   // One irrigation event is a volume-bounded batch. The pre-flush and
   // post-flush sections use only carrier water; metering pumps run only in
   // the middle FERTIGATE section. A zero volume SP preserves continuous
   // manual commissioning behavior.
   #Pre_Flush_Ratio_Limited := "DB1".Pre_Flush_Ratio;
   IF #Pre_Flush_Ratio_Limited < 0.0 THEN #Pre_Flush_Ratio_Limited := 0.0; END_IF;
   IF #Pre_Flush_Ratio_Limited > 1.0 THEN #Pre_Flush_Ratio_Limited := 1.0; END_IF;
   #Post_Flush_Ratio_Limited := "DB1".Post_Flush_Ratio;
   IF #Post_Flush_Ratio_Limited < 0.0 THEN #Post_Flush_Ratio_Limited := 0.0; END_IF;
   IF #Post_Flush_Ratio_Limited > (1.0 - #Pre_Flush_Ratio_Limited) THEN
      #Post_Flush_Ratio_Limited := 1.0 - #Pre_Flush_Ratio_Limited;
   END_IF;
   "DB1".Pre_Flush_Volume := "DB1".Water_Volume_SP * #Pre_Flush_Ratio_Limited;
   "DB1".Fertigation_End_Volume := "DB1".Water_Volume_SP
      * (1.0 - #Post_Flush_Ratio_Limited);
   "DB1".Batch_Fertigation_Active := FALSE;
   "DB1".Water_Batch_Active := FALSE;

   IF "DB1".Water_Enable < 0.5 THEN
      IF "DB1".Water_Volume_Complete THEN
         "DB1".Water_Batch_Phase := 4;
      ELSE
         "DB1".Water_Batch_Phase := 0;
      END_IF;
   ELSIF "DB1".Water_Volume_Complete THEN
      "DB1".Water_Batch_Phase := 4;
   ELSIF "DB1".Water_Volume_SP <= 0.0 THEN
      "DB1".Water_Batch_Phase := 2;
      "DB1".Water_Batch_Active := TRUE;
      "DB1".Batch_Fertigation_Active := "DB1".Water_Flow_OK;
   ELSIF "DB1".Water_Volume_Actual < "DB1".Pre_Flush_Volume THEN
      "DB1".Water_Batch_Phase := 1;
      "DB1".Water_Batch_Active := TRUE;
   ELSIF "DB1".Water_Volume_Actual < "DB1".Fertigation_End_Volume THEN
      "DB1".Water_Batch_Phase := 2;
      "DB1".Water_Batch_Active := TRUE;
      "DB1".Batch_Fertigation_Active := "DB1".Water_Flow_OK;
   ELSE
      "DB1".Water_Batch_Phase := 3;
      "DB1".Water_Batch_Active := TRUE;
   END_IF;

   // Scheme B: independent N, P, K and acid metering pumps.
   // Execution_Enable is FALSE by default, so legacy simulation behavior is isolated.
   "DB_Pump_N"(
      Enable := "DB_Actuator".Execution_Enable AND "DB1".Batch_Fertigation_Active
         AND NOT "DB1".Emergency_Stop,
      Flow_SP := "DB1".q_n_cmd,
      Flow_PV := "DB_Actuator".N_Flow_PV,
      Flow_Min := "DB_Actuator".N_Flow_Min,
      Flow_Max := "DB_Actuator".N_Flow_Max,
      AO_Off_Raw := "DB_Actuator".N_AO_Off_Raw,
      AO_Raw_Min := "DB_Actuator".N_AO_Raw_Min,
      AO_Raw_Max := "DB_Actuator".N_AO_Raw_Max,
      Kp_Flow := "DB_Actuator".N_Kp_Flow,
      Ki_Flow := "DB_Actuator".N_Ki_Flow,
      Cycle_Time_s := "DB_Actuator".Cycle_Time_s,
      Run_Feedback := "DB_Actuator".N_Run_Feedback,
      Drive_Ready := "DB_Actuator".N_Drive_Ready,
      Drive_Fault := "DB_Actuator".N_Drive_Fault,
      Tank_Low_Level := "DB_Actuator".N_Tank_Low_Level,
      Water_Flow_OK := "DB_Actuator".Water_Flow_OK,
      Reset := "DB_Actuator".Reset_All OR "DB_Actuator".N_Reset,
      Start_Fail_Delay_s := "DB_Actuator".N_Start_Fail_Delay_s,
      No_Flow_Delay_s := "DB_Actuator".N_No_Flow_Delay_s,
      Flow_Deviation_Delay_s := "DB_Actuator".N_Flow_Deviation_Delay_s,
      No_Flow_Threshold := "DB_Actuator".N_No_Flow_Threshold,
      Flow_Deviation_Abs := "DB_Actuator".N_Flow_Deviation_Abs,
      Flow_Deviation_Rel := "DB_Actuator".N_Flow_Deviation_Rel,
      Run_Command => "DB_Actuator".N_Run_Command,
      AO_Command_Raw => "DB_Actuator".N_AO_Command_Raw,
      Flow_SP_Limited => "DB_Actuator".N_Flow_SP_Limited,
      Running => "DB_Actuator".N_Running,
      Ready => "DB_Actuator".N_Ready,
      No_Flow_Alarm => "DB_Actuator".N_No_Flow_Alarm,
      Flow_Deviation_Alarm => "DB_Actuator".N_Flow_Deviation_Alarm,
      Start_Fail_Alarm => "DB_Actuator".N_Start_Fail_Alarm,
      Saturated => "DB_Actuator".N_Saturated,
      Interlocked => "DB_Actuator".N_Interlocked,
      Control_Percent => "DB_Actuator".N_Control_Percent
   );

   "DB_Pump_P"(
      Enable := "DB_Actuator".Execution_Enable AND "DB1".Batch_Fertigation_Active
         AND NOT "DB1".Emergency_Stop,
      Flow_SP := "DB1".q_p_cmd,
      Flow_PV := "DB_Actuator".P_Flow_PV,
      Flow_Min := "DB_Actuator".P_Flow_Min,
      Flow_Max := "DB_Actuator".P_Flow_Max,
      AO_Off_Raw := "DB_Actuator".P_AO_Off_Raw,
      AO_Raw_Min := "DB_Actuator".P_AO_Raw_Min,
      AO_Raw_Max := "DB_Actuator".P_AO_Raw_Max,
      Kp_Flow := "DB_Actuator".P_Kp_Flow,
      Ki_Flow := "DB_Actuator".P_Ki_Flow,
      Cycle_Time_s := "DB_Actuator".Cycle_Time_s,
      Run_Feedback := "DB_Actuator".P_Run_Feedback,
      Drive_Ready := "DB_Actuator".P_Drive_Ready,
      Drive_Fault := "DB_Actuator".P_Drive_Fault,
      Tank_Low_Level := "DB_Actuator".P_Tank_Low_Level,
      Water_Flow_OK := "DB_Actuator".Water_Flow_OK,
      Reset := "DB_Actuator".Reset_All OR "DB_Actuator".P_Reset,
      Start_Fail_Delay_s := "DB_Actuator".P_Start_Fail_Delay_s,
      No_Flow_Delay_s := "DB_Actuator".P_No_Flow_Delay_s,
      Flow_Deviation_Delay_s := "DB_Actuator".P_Flow_Deviation_Delay_s,
      No_Flow_Threshold := "DB_Actuator".P_No_Flow_Threshold,
      Flow_Deviation_Abs := "DB_Actuator".P_Flow_Deviation_Abs,
      Flow_Deviation_Rel := "DB_Actuator".P_Flow_Deviation_Rel,
      Run_Command => "DB_Actuator".P_Run_Command,
      AO_Command_Raw => "DB_Actuator".P_AO_Command_Raw,
      Flow_SP_Limited => "DB_Actuator".P_Flow_SP_Limited,
      Running => "DB_Actuator".P_Running,
      Ready => "DB_Actuator".P_Ready,
      No_Flow_Alarm => "DB_Actuator".P_No_Flow_Alarm,
      Flow_Deviation_Alarm => "DB_Actuator".P_Flow_Deviation_Alarm,
      Start_Fail_Alarm => "DB_Actuator".P_Start_Fail_Alarm,
      Saturated => "DB_Actuator".P_Saturated,
      Interlocked => "DB_Actuator".P_Interlocked,
      Control_Percent => "DB_Actuator".P_Control_Percent
   );

   "DB_Pump_K"(
      Enable := "DB_Actuator".Execution_Enable AND "DB1".Batch_Fertigation_Active
         AND NOT "DB1".Emergency_Stop,
      Flow_SP := "DB1".q_k_cmd,
      Flow_PV := "DB_Actuator".K_Flow_PV,
      Flow_Min := "DB_Actuator".K_Flow_Min,
      Flow_Max := "DB_Actuator".K_Flow_Max,
      AO_Off_Raw := "DB_Actuator".K_AO_Off_Raw,
      AO_Raw_Min := "DB_Actuator".K_AO_Raw_Min,
      AO_Raw_Max := "DB_Actuator".K_AO_Raw_Max,
      Kp_Flow := "DB_Actuator".K_Kp_Flow,
      Ki_Flow := "DB_Actuator".K_Ki_Flow,
      Cycle_Time_s := "DB_Actuator".Cycle_Time_s,
      Run_Feedback := "DB_Actuator".K_Run_Feedback,
      Drive_Ready := "DB_Actuator".K_Drive_Ready,
      Drive_Fault := "DB_Actuator".K_Drive_Fault,
      Tank_Low_Level := "DB_Actuator".K_Tank_Low_Level,
      Water_Flow_OK := "DB_Actuator".Water_Flow_OK,
      Reset := "DB_Actuator".Reset_All OR "DB_Actuator".K_Reset,
      Start_Fail_Delay_s := "DB_Actuator".K_Start_Fail_Delay_s,
      No_Flow_Delay_s := "DB_Actuator".K_No_Flow_Delay_s,
      Flow_Deviation_Delay_s := "DB_Actuator".K_Flow_Deviation_Delay_s,
      No_Flow_Threshold := "DB_Actuator".K_No_Flow_Threshold,
      Flow_Deviation_Abs := "DB_Actuator".K_Flow_Deviation_Abs,
      Flow_Deviation_Rel := "DB_Actuator".K_Flow_Deviation_Rel,
      Run_Command => "DB_Actuator".K_Run_Command,
      AO_Command_Raw => "DB_Actuator".K_AO_Command_Raw,
      Flow_SP_Limited => "DB_Actuator".K_Flow_SP_Limited,
      Running => "DB_Actuator".K_Running,
      Ready => "DB_Actuator".K_Ready,
      No_Flow_Alarm => "DB_Actuator".K_No_Flow_Alarm,
      Flow_Deviation_Alarm => "DB_Actuator".K_Flow_Deviation_Alarm,
      Start_Fail_Alarm => "DB_Actuator".K_Start_Fail_Alarm,
      Saturated => "DB_Actuator".K_Saturated,
      Interlocked => "DB_Actuator".K_Interlocked,
      Control_Percent => "DB_Actuator".K_Control_Percent
   );

   "DB_Pump_Acid"(
      Enable := "DB_Actuator".Execution_Enable AND "DB1".Batch_Fertigation_Active
         AND NOT "DB1".Emergency_Stop,
      Flow_SP := "DB1".q_a_cmd,
      Flow_PV := "DB_Actuator".Acid_Flow_PV,
      Flow_Min := "DB_Actuator".Acid_Flow_Min,
      Flow_Max := "DB_Actuator".Acid_Flow_Max,
      AO_Off_Raw := "DB_Actuator".Acid_AO_Off_Raw,
      AO_Raw_Min := "DB_Actuator".Acid_AO_Raw_Min,
      AO_Raw_Max := "DB_Actuator".Acid_AO_Raw_Max,
      Kp_Flow := "DB_Actuator".Acid_Kp_Flow,
      Ki_Flow := "DB_Actuator".Acid_Ki_Flow,
      Cycle_Time_s := "DB_Actuator".Cycle_Time_s,
      Run_Feedback := "DB_Actuator".Acid_Run_Feedback,
      Drive_Ready := "DB_Actuator".Acid_Drive_Ready,
      Drive_Fault := "DB_Actuator".Acid_Drive_Fault,
      Tank_Low_Level := "DB_Actuator".Acid_Tank_Low_Level,
      Water_Flow_OK := "DB_Actuator".Water_Flow_OK,
      Reset := "DB_Actuator".Reset_All OR "DB_Actuator".Acid_Reset,
      Start_Fail_Delay_s := "DB_Actuator".Acid_Start_Fail_Delay_s,
      No_Flow_Delay_s := "DB_Actuator".Acid_No_Flow_Delay_s,
      Flow_Deviation_Delay_s := "DB_Actuator".Acid_Flow_Deviation_Delay_s,
      No_Flow_Threshold := "DB_Actuator".Acid_No_Flow_Threshold,
      Flow_Deviation_Abs := "DB_Actuator".Acid_Flow_Deviation_Abs,
      Flow_Deviation_Rel := "DB_Actuator".Acid_Flow_Deviation_Rel,
      Run_Command => "DB_Actuator".Acid_Run_Command,
      AO_Command_Raw => "DB_Actuator".Acid_AO_Command_Raw,
      Flow_SP_Limited => "DB_Actuator".Acid_Flow_SP_Limited,
      Running => "DB_Actuator".Acid_Running,
      Ready => "DB_Actuator".Acid_Ready,
      No_Flow_Alarm => "DB_Actuator".Acid_No_Flow_Alarm,
      Flow_Deviation_Alarm => "DB_Actuator".Acid_Flow_Deviation_Alarm,
      Start_Fail_Alarm => "DB_Actuator".Acid_Start_Fail_Alarm,
      Saturated => "DB_Actuator".Acid_Saturated,
      Interlocked => "DB_Actuator".Acid_Interlocked,
      Control_Percent => "DB_Actuator".Acid_Control_Percent
   );

   "DB_Actuator".Any_Demand := "DB_Actuator".Execution_Enable
      AND "DB1".Batch_Fertigation_Active AND (
      ("DB1".q_n_cmd > 0.0) OR ("DB1".q_p_cmd > 0.0)
      OR ("DB1".q_k_cmd > 0.0) OR ("DB1".q_a_cmd > 0.0));

   "DB_Actuator".Any_Trip := "DB_Actuator".Execution_Enable AND (
      "DB1".Water_Pump_Fault
      OR
      "DB_Actuator".N_Start_Fail_Alarm OR "DB_Actuator".N_No_Flow_Alarm
      OR "DB_Actuator".P_Start_Fail_Alarm OR "DB_Actuator".P_No_Flow_Alarm
      OR "DB_Actuator".K_Start_Fail_Alarm OR "DB_Actuator".K_No_Flow_Alarm
      OR "DB_Actuator".Acid_Start_Fail_Alarm OR "DB_Actuator".Acid_No_Flow_Alarm
      OR "DB_Actuator".N_Drive_Fault OR "DB_Actuator".P_Drive_Fault
      OR "DB_Actuator".K_Drive_Fault OR "DB_Actuator".Acid_Drive_Fault
      OR "DB_Actuator".N_Tank_Low_Level OR "DB_Actuator".P_Tank_Low_Level
      OR "DB_Actuator".K_Tank_Low_Level OR "DB_Actuator".Acid_Tank_Low_Level
      OR ("DB_Actuator".Any_Demand AND NOT "DB_Actuator".Water_Flow_OK));

   "DB_Actuator".Any_Alarm := "DB_Actuator".Execution_Enable AND (
      "DB_Actuator".Any_Trip OR "DB1".Water_Pump_Alarm
      OR "DB_Actuator".N_Flow_Deviation_Alarm
      OR "DB_Actuator".P_Flow_Deviation_Alarm
      OR "DB_Actuator".K_Flow_Deviation_Alarm
      OR "DB_Actuator".Acid_Flow_Deviation_Alarm);

   "DB1".Actuator_Execution_Enable := "DB_Actuator".Execution_Enable;
   "DB1".Actuator_Any_Alarm := "DB_Actuator".Any_Alarm;
   "DB1".Actuator_Any_Trip := "DB_Actuator".Any_Trip;

   IF "DB_Actuator".Execution_Enable THEN
      // The total fertilizer AO is forced off in Scheme B to prevent double dosing.
      "DB1".AQ_Valve_F_Raw := 0;
      "DB1".AQ_Valve_N_Raw := "DB_Actuator".N_AO_Command_Raw;
      "DB1".AQ_Valve_P_Raw := "DB_Actuator".P_AO_Command_Raw;
      "DB1".AQ_Valve_K_Raw := "DB_Actuator".K_AO_Command_Raw;
      "DB1".AQ_Valve_A_Raw := "DB_Actuator".Acid_AO_Command_Raw;

      // Real feedback replaces the previous command-as-feedback simulation value.
      "DB1".Valve_F_Actual := "DB_Actuator".N_Flow_PV
         + "DB_Actuator".P_Flow_PV + "DB_Actuator".K_Flow_PV;
      "DB1".Valve_A_Actual := "DB_Actuator".Acid_Flow_PV;
   END_IF;

   IF "DB1".System_Alarm_Reset THEN
      "DB1".System_Alarm_Light := FALSE;
   END_IF;
   IF "DB_Actuator".Any_Alarm THEN
      "DB1".System_Alarm_Light := TRUE;
   END_IF;
END_FUNCTION

FUNCTION "FC_CallFertigationControl" : Void
{ S7_Optimized_Access := 'TRUE' }
VERSION : 0.1
   VAR_TEMP
      Mode_EStop : Bool;
      Mode_Manual : Bool;
      Mode_Remote_Auto : Bool;
      Mode_Stage_Auto : Bool;
      Mode_Local_Auto : Bool;
      Mode_Standby : Bool;
      Remote_Auto_Available : Bool;
      PID_Control_Enable : Bool;
      Gain_Desired_Point : Int;
      Gain_q_f_Estimate : Real;
      Effective_Decoupler_Enable : Bool;
      Control_CycleTime : Real;
   END_VAR

BEGIN
   // 在 OB1 中调用本 FC，即可完成：
   // DB1 输入区 -> FB_FertigationControl -> DB1 输出区。
   // 固定模式表：
   // 1) Emergency_Stop=TRUE -> 急停，所有输出归零。
   // 2) Emergency_Stop=FALSE 且 Manual_Mode=TRUE -> 手动直接流量输出。
   // 3) Emergency_Stop=FALSE 且 Manual_Mode=FALSE 且 Auto_Mode=TRUE 且 SAC_Enable=TRUE -> 远程自动。
   // 4) Emergency_Stop=FALSE 且 Manual_Mode=FALSE 且 Auto_Mode=TRUE 且 SAC_Enable=FALSE 且 Stage_Auto_SP_Enable=TRUE -> 阶段自动。
   // 5) Emergency_Stop=FALSE 且 Manual_Mode=FALSE 且 Auto_Mode=TRUE 且 SAC_Enable=FALSE 且 Stage_Auto_SP_Enable=FALSE -> 本地定值自动。
   // 6) Emergency_Stop=FALSE 且 Manual_Mode=FALSE 且 Auto_Mode=FALSE -> 待机，所有输出归零。
   // 开关量联锁和报警灯由 FC_ModeInterlock_LAD 完成。
   // 六种互斥运行模式由 FC_ModeSelector_LAD 完成。
   // 连续量限幅、斜坡、模拟量换算和自动控制算法保留在 SCL。

   "FC_ModeInterlock_LAD"();

   // 远程命令只有在心跳正常时才有效；失联后把 SAC 请求视为无效，
   // 由现有 LAD 模式表自动选择阶段自动或本地定值自动。
   IF NOT "DB1".Remote_Comms_OK THEN
      "DB1".SAC_Enable := FALSE;
   END_IF;
   // 自动模式的本地来源固定为生长阶段目标，不提供人工来源切换。
   "DB1".Stage_Auto_SP_Enable := TRUE;
   #Remote_Auto_Available := "DB1".SAC_Enable AND "DB1".Remote_Comms_OK;

   "FC_ModeSelector_LAD"(
      Emergency_Stop := "DB1".Emergency_Stop,
      Manual_Mode := "DB1".Manual_Mode,
      Auto_Mode := "DB1".Auto_Mode,
      SAC_Enable := #Remote_Auto_Available,
      Stage_Auto_SP_Enable := "DB1".Stage_Auto_SP_Enable,
      Mode_EStop => #Mode_EStop,
      Mode_Manual => #Mode_Manual,
      Mode_Remote_Auto => #Mode_Remote_Auto,
      Mode_Stage_Auto => #Mode_Stage_Auto,
      Mode_Local_Auto => #Mode_Local_Auto,
      Mode_Standby => #Mode_Standby
   );

   // Manual_Active, Auto_Active, Manual_PumpValve_Enable and the two manual
   // flow selections are discrete interlocks owned by FC_ModeInterlock_LAD.
   // Do not assign them again in SCL; one tag must have one logic owner.

   #PID_Control_Enable := #Mode_Manual OR #Mode_Remote_Auto OR #Mode_Stage_Auto OR #Mode_Local_Auto;

   // PLC-native low/medium/high gain schedule. Python only commissions the
   // table; normal selection, hysteresis and bumpless handoff run in the CPU.
   "DB1".Gain_Schedule_Valid := "DB1".Gain_Low_Valid
      AND "DB1".Gain_Mid_Valid AND "DB1".Gain_High_Valid
      AND ("DB1".Gain_Low_G_EC_F > 0.000001) AND ("DB1".Gain_Low_G_pH_A < -0.000001)
      AND ("DB1".Gain_Mid_G_EC_F > 0.000001) AND ("DB1".Gain_Mid_G_pH_A < -0.000001)
      AND ("DB1".Gain_High_G_EC_F > 0.000001) AND ("DB1".Gain_High_G_pH_A < -0.000001)
      AND ("DB1".Gain_Low_EC_SP > 0.0)
      AND ("DB1".Gain_Mid_EC_SP > 0.0)
      AND ("DB1".Gain_High_EC_SP > 0.0)
      AND ("DB1".Gain_Low_q_f < "DB1".Gain_Mid_q_f)
      AND ("DB1".Gain_Mid_q_f < "DB1".Gain_High_q_f)
      AND ("DB1".Gain_LM_Threshold < "DB1".Gain_MH_Threshold)
      AND ("DB1".Gain_Schedule_Hysteresis >= 0.0)
      AND ("DB1".Gain_Min_Hold_s >= 0.0);

   IF ("DB1".EC_Set_SP > 0.0) AND ("DB1".EC_Set_SP < 34.0) THEN
      #Gain_q_f_Estimate := ("DB1".EC_Set_SP * 136.0) / (35.0 - "DB1".EC_Set_SP);
   ELSE
      #Gain_q_f_Estimate := 0.0;
   END_IF;
   IF ("DB1".Gain_Point_Override >= 0) AND ("DB1".Gain_Point_Override <= 2) THEN
      #Gain_Desired_Point := "DB1".Gain_Point_Override;
   ELSIF "DB1".Active_Gain_Point = 0 THEN
      IF #Gain_q_f_Estimate > ("DB1".Gain_LM_Threshold + "DB1".Gain_Schedule_Hysteresis) THEN
         #Gain_Desired_Point := 1;
      ELSE
         #Gain_Desired_Point := 0;
      END_IF;
   ELSIF "DB1".Active_Gain_Point = 2 THEN
      IF #Gain_q_f_Estimate < ("DB1".Gain_MH_Threshold - "DB1".Gain_Schedule_Hysteresis) THEN
         #Gain_Desired_Point := 1;
      ELSE
         #Gain_Desired_Point := 2;
      END_IF;
   ELSE
      IF #Gain_q_f_Estimate < ("DB1".Gain_LM_Threshold - "DB1".Gain_Schedule_Hysteresis) THEN
         #Gain_Desired_Point := 0;
      ELSIF #Gain_q_f_Estimate > ("DB1".Gain_MH_Threshold + "DB1".Gain_Schedule_Hysteresis) THEN
         #Gain_Desired_Point := 2;
      ELSE
         #Gain_Desired_Point := 1;
      END_IF;
   END_IF;

   IF "DB1".Gain_Schedule_Enable AND "DB1".Gain_Schedule_Valid THEN
      IF "DB1".Gain_Hold_Elapsed_s < 3600.0 THEN
         "DB1".Gain_Hold_Elapsed_s := "DB1".Gain_Hold_Elapsed_s + 0.1;
      END_IF;
      IF "DB1".Active_Gain_Point < 0 THEN
         "DB1".Gain_Switch_Pending := TRUE;
      ELSIF (#Gain_Desired_Point <> "DB1".Active_Gain_Point)
         AND ("DB1".Gain_Hold_Elapsed_s >= "DB1".Gain_Min_Hold_s) THEN
         "DB1".Gain_Switch_Pending := TRUE;
      END_IF;

      // Pending makes the effective enable FALSE below. The FB ramps its
      // applied weight to zero before this block replaces the active matrix.
      IF "DB1".Gain_Switch_Pending AND ("DB1".Decoupler_Weight_Applied <= 0.01) THEN
         IF #Gain_Desired_Point = 0 THEN
            "DB1".G_EC_F := "DB1".Gain_Low_G_EC_F;
            "DB1".G_EC_A := "DB1".Gain_Low_G_EC_A;
            "DB1".G_pH_F := "DB1".Gain_Low_G_pH_F;
            "DB1".G_pH_A := "DB1".Gain_Low_G_pH_A;
            "DB1".IMC_Tau_EC_s := "DB1".Gain_Low_Tau_s;
            "DB1".IMC_Delay_s := "DB1".Gain_Low_Delay_s;
            "DB1".Mixing_Delay_s := "DB1".Gain_Low_Delay_s;
            "DB1".Active_Gain_EC_SP := "DB1".Gain_Low_EC_SP;
            "DB1".Active_Gain_q_f := "DB1".Gain_Low_q_f;
         ELSIF #Gain_Desired_Point = 1 THEN
            "DB1".G_EC_F := "DB1".Gain_Mid_G_EC_F;
            "DB1".G_EC_A := "DB1".Gain_Mid_G_EC_A;
            "DB1".G_pH_F := "DB1".Gain_Mid_G_pH_F;
            "DB1".G_pH_A := "DB1".Gain_Mid_G_pH_A;
            "DB1".IMC_Tau_EC_s := "DB1".Gain_Mid_Tau_s;
            "DB1".IMC_Delay_s := "DB1".Gain_Mid_Delay_s;
            "DB1".Mixing_Delay_s := "DB1".Gain_Mid_Delay_s;
            "DB1".Active_Gain_EC_SP := "DB1".Gain_Mid_EC_SP;
            "DB1".Active_Gain_q_f := "DB1".Gain_Mid_q_f;
         ELSE
            "DB1".G_EC_F := "DB1".Gain_High_G_EC_F;
            "DB1".G_EC_A := "DB1".Gain_High_G_EC_A;
            "DB1".G_pH_F := "DB1".Gain_High_G_pH_F;
            "DB1".G_pH_A := "DB1".Gain_High_G_pH_A;
            "DB1".IMC_Tau_EC_s := "DB1".Gain_High_Tau_s;
            "DB1".IMC_Delay_s := "DB1".Gain_High_Delay_s;
            "DB1".Mixing_Delay_s := "DB1".Gain_High_Delay_s;
            "DB1".Active_Gain_EC_SP := "DB1".Gain_High_EC_SP;
            "DB1".Active_Gain_q_f := "DB1".Gain_High_q_f;
         END_IF;
         "DB1".Active_Gain_Point := #Gain_Desired_Point;
         "DB1".Gain_Hold_Elapsed_s := 0.0;
         "DB1".Gain_Switch_Pending := FALSE;
      END_IF;
   ELSE
      "DB1".Gain_Switch_Pending := FALSE;
      "DB1".Gain_Hold_Elapsed_s := 0.0;
   END_IF;

   // Validate the decoupling contract before any mode-specific early return.
   // This keeps DB1 diagnostics current while the PLC is in standby or E-stop.
   "DB1".Decoupler_Determinant := "DB1".G_EC_F * "DB1".G_pH_A
      - "DB1".G_EC_A * "DB1".G_pH_F;
   "DB1".Decoupler_Valid := ("DB1".Decoupler_Determinant_Min > 0.0)
      AND (ABS("DB1".Decoupler_Determinant) >= "DB1".Decoupler_Determinant_Min)
      AND ("DB1".G_EC_F > 0.000001)
      AND ("DB1".G_pH_A < -0.000001)
      AND ("DB1".Decoupler_Weight >= 0.0)
      AND ("DB1".Decoupler_Weight <= 1.0)
      AND ("DB1".Decoupler_Regularization >= 0.0)
      AND ("DB1".Decoupler_Regularization <= 1.0)
      AND ("DB1".Mixing_Delay_s >= 0.0)
      AND ("DB1".Mixing_Delay_s <= 600.0)
      AND ("DB1".q_f_max > "DB1".q_f_min)
      AND ("DB1".q_a_max > "DB1".q_a_min);
   IF "DB1".Decoupler_Enable AND NOT "DB1".Decoupler_Valid THEN
      "DB1".Decoupler_Enable := FALSE;
   END_IF;
   #Effective_Decoupler_Enable := "DB1".Decoupler_Enable
      AND ("DB1".Controller_Mode = 2)
      AND NOT "DB1".Gain_Switch_Pending
      AND ("DB1".E4_Approved OR ("DB1".E4_Test_Enable AND "DB1".Remote_Comms_OK));
   "DB1".Decoupler_Active_Diag := #Effective_Decoupler_Enable AND "DB1".Decoupler_Valid;

   IF #Mode_EStop THEN
      "DB1".q_f_cmd := 0.0;
      "DB1".q_a_cmd := 0.0;
      "DB1".q_n_cmd := 0.0;
      "DB1".q_p_cmd := 0.0;
      "DB1".q_k_cmd := 0.0;
      "DB1".Valve_F_Actual := 0.0;
      "DB1".Valve_A_Actual := 0.0;
      "DB1".AQ_Valve_F_Raw := 0;
      "DB1".AQ_Valve_A_Raw := 0;
      "DB1".AQ_Valve_N_Raw := 0;
      "DB1".AQ_Valve_P_Raw := 0;
      "DB1".AQ_Valve_K_Raw := 0;
      "DB1".Actual_Valve_F := 0.0;
      "DB1".Actual_Valve_A := 0.0;
      "DB1".Valve_F_Opt_SP := 0.0;
      "DB1".Valve_A_Opt_SP := 0.0;
      "DB1".Ramp_Target_F := 0.0;
      "DB1".Ramp_Target_A := 0.0;
      RETURN;
   END_IF;

   // 待机没有任何目标来源，所有执行量安全归零。
   IF #Mode_Standby THEN
      "DB1".q_f_cmd := 0.0;
      "DB1".q_a_cmd := 0.0;
      "DB1".q_n_cmd := 0.0;
      "DB1".q_p_cmd := 0.0;
      "DB1".q_k_cmd := 0.0;
      "DB1".Valve_F_Actual := 0.0;
      "DB1".Valve_A_Actual := 0.0;
      "DB1".AQ_Valve_F_Raw := 0;
      "DB1".AQ_Valve_A_Raw := 0;
      "DB1".AQ_Valve_N_Raw := 0;
      "DB1".AQ_Valve_P_Raw := 0;
      "DB1".AQ_Valve_K_Raw := 0;
      "DB1".Actual_Valve_F := 0.0;
      "DB1".Actual_Valve_A := 0.0;
      "DB1".Valve_F_Opt_SP := 0.0;
      "DB1".Valve_A_Opt_SP := 0.0;
      "DB1".Ramp_Target_F := 0.0;
      "DB1".Ramp_Target_A := 0.0;
      RETURN;
   END_IF;

   // Remote residual command: clamp first, then resolve the absolute EC target.
   // Legacy HMIs may still write EC_Set_SP directly when residual fields are 0.
   IF #Mode_Remote_Auto THEN
      IF "DB1".Water_Multiplier_SP < 0.8 THEN "DB1".Water_Multiplier_SP := 0.8; END_IF;
      IF "DB1".Water_Multiplier_SP > 1.2 THEN "DB1".Water_Multiplier_SP := 1.2; END_IF;
      IF "DB1".EC_Residual_SP < -0.15 THEN "DB1".EC_Residual_SP := -0.15; END_IF;
      IF "DB1".EC_Residual_SP > 0.15 THEN "DB1".EC_Residual_SP := 0.15; END_IF;
      IF "DB1".Growth_Stage = 0 THEN
         "DB1".EC_Set_SP := 0.8 + "DB1".EC_Residual_SP;
      ELSIF "DB1".Growth_Stage = 1 THEN
         "DB1".EC_Set_SP := 1.1 + "DB1".EC_Residual_SP;
      ELSIF "DB1".Growth_Stage = 2 THEN
         "DB1".EC_Set_SP := 1.5 + "DB1".EC_Residual_SP;
      ELSE
         "DB1".EC_Set_SP := 1.0 + "DB1".EC_Residual_SP;
      END_IF;
      "DB1".pH_Set_SP := ("DB1".pH_Band_Low + "DB1".pH_Band_High) * 0.5;
      IF "DB1".Batch_Water_Target_L > 0.0 THEN
         "DB1".Water_Volume_SP := "DB1".Batch_Water_Target_L;
      END_IF;
   END_IF;

   IF #Mode_Stage_Auto THEN
      IF "DB1".Growth_Stage = 0 THEN
         "DB1".EC_Set_SP := 0.8;
         "DB1".pH_Set_SP := 6.2;
      ELSIF "DB1".Growth_Stage = 1 THEN
         "DB1".EC_Set_SP := 1.1;
         "DB1".pH_Set_SP := 6.1;
      ELSIF "DB1".Growth_Stage = 2 THEN
         "DB1".EC_Set_SP := 1.5;
         "DB1".pH_Set_SP := 5.9;
      ELSE
         "DB1".EC_Set_SP := 1.0;
         "DB1".pH_Set_SP := 6.1;
      END_IF;
   END_IF;

   // 真实设备没有 N/P/K 在线反馈时，只使用 PLC 内置阶段配方。
   // PLCSIM/Python 置 NPK_Feedback_Valid 后保留脚本写入的目标和土壤反馈。
   IF NOT ("DB1".NPK_Feedback_Valid AND "DB1".Remote_Comms_OK) THEN
      IF "DB1".Growth_Stage = 0 THEN
         "DB1".N_Target := 0.75; "DB1".P_Target := 0.55; "DB1".K_Target := 0.65;
      ELSIF "DB1".Growth_Stage = 1 THEN
         "DB1".N_Target := 0.95; "DB1".P_Target := 0.75; "DB1".K_Target := 0.90;
      ELSIF "DB1".Growth_Stage = 2 THEN
         "DB1".N_Target := 1.10; "DB1".P_Target := 0.85; "DB1".K_Target := 1.25;
      ELSE
         "DB1".N_Target := 0.85; "DB1".P_Target := 0.65; "DB1".K_Target := 1.05;
      END_IF;
   END_IF;

   // Accelerated E4 HIL advances controller dynamics once per new Python
   // heartbeat. Hardware and all normal PLC modes keep the real 0.1 s cycle.
   IF "DB1".E4_Test_Enable AND "DB1".E4_Compressed_Time_Enable
      AND ("DB1".E4_Sim_Step_s >= 0.1) AND ("DB1".E4_Sim_Step_s <= 300.0) THEN
      #Control_CycleTime := "DB1".E4_Sim_Step_s;
   ELSE
      #Control_CycleTime := 0.1;
   END_IF;

   "inst_FertigationControl"(
      EC_Set_SP := "DB1".EC_Set_SP,
      pH_Set_SP := "DB1".pH_Set_SP,
      EC_Actual := "DB1".EC_Actual,
      pH_Actual := "DB1".pH_Actual,
      SAC_Enable := #PID_Control_Enable,
      Remote_Comms_Required := #Mode_Remote_Auto,
      Local_Fallback_Mode := (#Mode_Manual OR #Mode_Stage_Auto OR #Mode_Local_Auto),
      Local_EC_Bias := 0.0,
      Local_pH_Bias := 0.0,
      Remote_Heartbeat := "DB1".Remote_Heartbeat,
      CycleTime := #Control_CycleTime,
      E4_Compressed_Timing_Enable := "DB1".E4_Test_Enable
         AND "DB1".E4_Compressed_Time_Enable,
      Kp_EC := "DB1".Kp_EC_Set,
      Ki_EC := "DB1".Ki_EC_Set,
      Kd_EC := "DB1".Kd_EC_Set,
      Kp_pH := "DB1".Kp_pH_Set,
      Ki_pH := "DB1".Ki_pH_Set,
      Kd_pH := "DB1".Kd_pH_Set,
      EC_Filter_Tau := 2.0,
      pH_Filter_Tau := 4.0,
      EC_Deadband := 0.005,
      pH_Deadband := 0.005,
      EC_Trim_Band := "DB1".EC_Trim_Band,
      pH_Trim_Band := "DB1".pH_Trim_Band,
      EC_MaxInputStep := 0.15,
      pH_MaxInputStep := 0.10,
      q_f_min := "DB1".q_f_min,
      q_f_max := "DB1".q_f_max,
      q_a_min := "DB1".q_a_min,
      q_a_max := "DB1".q_a_max,
      Decoupler_Enable := #Effective_Decoupler_Enable,
      Decoupler_Valid := "DB1".Decoupler_Valid,
      G_EC_F := "DB1".G_EC_F,
      G_EC_A := "DB1".G_EC_A,
      G_pH_F := "DB1".G_pH_F,
      G_pH_A := "DB1".G_pH_A,
      Decoupler_Weight := "DB1".Decoupler_Weight,
      Decoupler_Regularization := "DB1".Decoupler_Regularization,
      Mixing_Delay_s := "DB1".Mixing_Delay_s,
      N_Enable := "DB1".N_Enable,
      N_Ratio := "DB1".N_Ratio,
      N_Target := "DB1".N_Target,
      N_Actual := "DB1".N_Actual,
      Kp_N := "DB1".Kp_N_Set,
      Ki_N := "DB1".Ki_N_Set,
      Kd_N := "DB1".Kd_N_Set,
      N_Max := "DB1".N_Max,
      P_Enable := "DB1".P_Enable,
      P_Ratio := "DB1".P_Ratio,
      P_Target := "DB1".P_Target,
      P_Actual := "DB1".P_Actual,
      Kp_P := "DB1".Kp_P_Set,
      Ki_P := "DB1".Ki_P_Set,
      Kd_P := "DB1".Kd_P_Set,
      P_Max := "DB1".P_Max,
      K_Enable := "DB1".K_Enable,
      K_Ratio := "DB1".K_Ratio,
      K_Target := "DB1".K_Target,
      K_Actual := "DB1".K_Actual,
      Kp_K := "DB1".Kp_K_Set,
      Ki_K := "DB1".Ki_K_Set,
      Kd_K := "DB1".Kd_K_Set,
      K_Max := "DB1".K_Max,
      Watchdog_Limit := 10000,
      Growth_Stage := "DB1".Growth_Stage,
      NPK_Feedback_Valid := "DB1".NPK_Feedback_Valid AND "DB1".Remote_Comms_OK,
      Compressed_HIL_Enable := "DB1".Compressed_HIL_Enable AND "DB1".Remote_Comms_OK,
      Fixed_PID_Test_Enable := "DB1".Fixed_PID_Test_Enable AND "DB1".Remote_Comms_OK,
      Controller_Mode := "DB1".Controller_Mode,
      pH_Band_Low := "DB1".pH_Band_Low,
      pH_Band_High := "DB1".pH_Band_High,
      pH_Pulse_On_s := "DB1".pH_Pulse_On_s,
      pH_Pulse_Off_s := "DB1".pH_Pulse_Off_s,
      pH_Pulse_Flow := "DB1".pH_Pulse_Flow,
      IMC_Lambda_EC_s := "DB1".IMC_Lambda_EC_s,
      IMC_Tau_EC_s := "DB1".IMC_Tau_EC_s,
      IMC_Delay_s := "DB1".IMC_Delay_s,
      IMC_EC_Operating_SP := "DB1".Active_Gain_EC_SP,
      IMC_q_f_Operating := "DB1".Active_Gain_q_f,
      Remote_Comms_OK => "DB1".Remote_Comms_OK,
      Watchdog_Timer => "DB1".Watchdog_Timer,
      Stage_EC_SP => "DB1".Stage_EC_SP,
      Stage_pH_SP => "DB1".Stage_pH_SP,
      Active_EC_SP => "DB1".Active_EC_SP,
      Active_pH_SP => "DB1".Active_pH_SP,
      Setpoint_Protection_Active => "DB1".Setpoint_Protection_Active,
      q_f_cmd => "DB1".q_f_cmd,
      q_a_cmd => "DB1".q_a_cmd,
      Valve_F_Actual => "DB1".Valve_F_Actual,
      Valve_A_Actual => "DB1".Valve_A_Actual,
      AQ_Valve_F_Raw => "DB1".AQ_Valve_F_Raw,
      AQ_Valve_A_Raw => "DB1".AQ_Valve_A_Raw,
      q_n_cmd => "DB1".q_n_cmd,
      q_p_cmd => "DB1".q_p_cmd,
      q_k_cmd => "DB1".q_k_cmd,
      AQ_Valve_N_Raw => "DB1".AQ_Valve_N_Raw,
      AQ_Valve_P_Raw => "DB1".AQ_Valve_P_Raw,
      AQ_Valve_K_Raw => "DB1".AQ_Valve_K_Raw,
      q_f_limited => "DB1".q_f_limited,
      q_a_limited => "DB1".q_a_limited,
      Kp_EC_Effective_Out => "DB1".Kp_EC_Effective,
      Ki_EC_Effective_Out => "DB1".Ki_EC_Effective,
      Kd_EC_Effective_Out => "DB1".Kd_EC_Effective,
      Kp_pH_Effective_Out => "DB1".Kp_pH_Effective,
      Ki_pH_Effective_Out => "DB1".Ki_pH_Effective,
      Kd_pH_Effective_Out => "DB1".Kd_pH_Effective,
      EC_PID_Error_Out => "DB1".EC_PID_Error,
      pH_PID_Error_Out => "DB1".pH_PID_Error,
      EC_PID_Integral_Out => "DB1".EC_PID_Integral,
      pH_PID_Integral_Out => "DB1".pH_PID_Integral,
      q_f_Feedforward_Out => "DB1".q_f_Feedforward,
      q_f_PID_Correction_Out => "DB1".q_f_PID_Correction,
      q_a_Feedforward_Out => "DB1".q_a_Feedforward,
      q_a_PID_Correction_Out => "DB1".q_a_PID_Correction,
      N_Error_Out => "DB1".N_Error,
      P_Error_Out => "DB1".P_Error,
      K_Error_Out => "DB1".K_Error,
      N_PID_Correction_Out => "DB1".N_PID_Correction,
      P_PID_Correction_Out => "DB1".P_PID_Correction,
      K_PID_Correction_Out => "DB1".K_PID_Correction,
      NPK_Optimization_Weight_Out => "DB1".NPK_Optimization_Weight,
      NPK_Capacity_Limited_Out => "DB1".NPK_Capacity_Limited,
      Feedforward_Hold_Active_Out => "DB1".Feedforward_Hold_Active,
      Adaptive_PID_Active_Out => "DB1".Adaptive_PID_Active,
      Delta_q_f_Out => "DB1".Delta_q_f,
      Delta_q_a_Out => "DB1".Delta_q_a,
      pH_Safety_Active_Out => "DB1".pH_Safety_Active,
      pH_Flush_Request_Out => "DB1".pH_Flush_Request,
      Batch_Reject_Out => "DB1".Batch_Reject,
      IMC_Smith_Active_Out => "DB1".IMC_Smith_Active,
      Smith_EC_Predicted_Out => "DB1".Smith_EC_Predicted,
      Decoupling_Limited_Out => "DB1".Decoupling_Limited,
      Decoupler_Weight_Applied_Out => "DB1".Decoupler_Weight_Applied
   );

   // Volume diagnostics are reset with the batch and integrated only while
   // the batch is active. Values are engineering-unit estimates until E1 pump
   // calibration replaces command flow with measured flow.
   "DB1".Water_Accumulated_L := "DB1".Water_Volume_Actual;
   IF "DB1".Water_Pump_Reset THEN
      "DB1".Fertilizer_Accumulated_L := 0.0;
      "DB1".Acid_Accumulated_L := 0.0;
   ELSIF "DB1".Water_Batch_Active THEN
      "DB1".Fertilizer_Accumulated_L := "DB1".Fertilizer_Accumulated_L
         + "DB1".q_f_cmd * 0.1 / 60.0;
      "DB1".Acid_Accumulated_L := "DB1".Acid_Accumulated_L
         + "DB1".q_a_cmd * 0.1 / 60.0;
   END_IF;

   // Manual commissioning bypasses EC/pH PID and writes the requested flow
   // values to the same bounded command variables used by the execution layer.
   // This is deliberately limited to Manual_Mode; automatic and SAC paths
   // remain entirely inside FB_FertigationControl.
   IF #Mode_Manual THEN
      "DB1".q_f_cmd := "DB1".Manual_q_f_Selected;
      IF "DB1".q_f_cmd < "DB1".q_f_min THEN "DB1".q_f_cmd := "DB1".q_f_min; END_IF;
      IF "DB1".q_f_cmd > "DB1".q_f_max THEN "DB1".q_f_cmd := "DB1".q_f_max; END_IF;
      "DB1".q_a_cmd := "DB1".Manual_q_a_Selected;
      IF "DB1".q_a_cmd < "DB1".q_a_min THEN "DB1".q_a_cmd := "DB1".q_a_min; END_IF;
      IF "DB1".q_a_cmd > "DB1".q_a_max THEN "DB1".q_a_cmd := "DB1".q_a_max; END_IF;
      "DB1".q_n_cmd := "DB1".Manual_q_n_Set;
      "DB1".q_p_cmd := "DB1".Manual_q_p_Set;
      "DB1".q_k_cmd := "DB1".Manual_q_k_Set;
      "DB1".q_f_limited := ("DB1".q_f_cmd <> "DB1".Manual_q_f_Selected);
      "DB1".q_a_limited := ("DB1".q_a_cmd <> "DB1".Manual_q_a_Selected);
      "DB1".q_f_raw := "DB1".Manual_q_f_Selected;
      "DB1".q_a_raw := "DB1".Manual_q_a_Selected;
   END_IF;

   // 测试反馈和压缩 HIL 标志在通信超时后自动恢复真实设备默认。
   IF NOT "DB1".Remote_Comms_OK THEN
      "DB1".NPK_Feedback_Valid := FALSE;
      "DB1".Compressed_HIL_Enable := FALSE;
      "DB1".Fixed_PID_Test_Enable := FALSE;
   END_IF;

   // 同步部分内部状态到 DB1，方便在线监控。
   // Execute the isolated real-actuator layer after the supervisory controller.
   "FC_CallDosingPumps"();

   "DB1".Last_Heartbeat := "inst_FertigationControl".Last_Heartbeat;
   "DB1".Watchdog_Count := "inst_FertigationControl".Watchdog_Count;
   "DB1".q_f_raw := "inst_FertigationControl".q_f_raw;
   "DB1".q_a_raw := "inst_FertigationControl".q_a_raw;

   // 兼容旧变量名，若旧监控画面或旧网络还在看 Actual_Valve_F/A，
   // 这里同步为当前 B 方案执行层输出。
   "DB1".Actual_Valve_F := "DB1".Valve_F_Actual;
   "DB1".Actual_Valve_A := "DB1".Valve_A_Actual;
   "DB1".Valve_F_Opt_SP := "DB1".q_f_cmd;
   "DB1".Valve_A_Opt_SP := "DB1".q_a_cmd;
   "DB1".Ramp_Target_F := "DB1".q_f_cmd;
   "DB1".Ramp_Target_A := "DB1".q_a_cmd;
   "DB1".Remote_Comms_Was_OK := "DB1".Remote_Comms_OK;
END_FUNCTION
